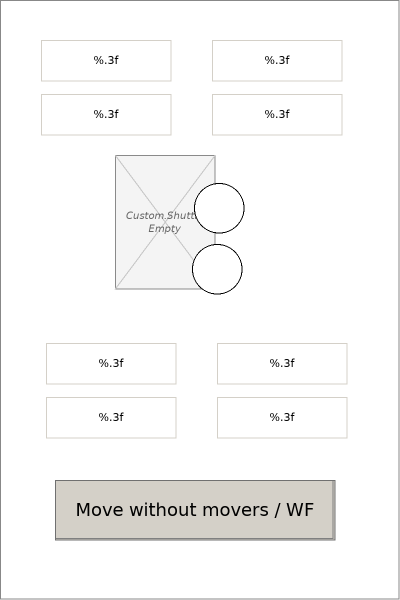
VISUALIZATION VISU_ST140  // 400x600
    Image (115,155 100x134), angle 90, invisible if: NOT __ISVALIDREF(GVL.st140_aut._Mover), image: Custom.Shuttle Empty
    Button (55,480 280x60), "Move without movers / WF", colour toggle: HMI.bArForceCyclusState[StationList_e.ST140]
        tap HMI.btArForceCyclus[StationList_e.ST140].button
    Ellipse (194,183 50x50)
    Ellipse (192,244 50x50)
    Textfield (41,40 130x41), "%.3f"
    Textfield (212,40 130x41), "%.3f"
    Textfield (212,94 130x41), "%.3f"
    Textfield (46,343 130x41), "%.3f"
    Textfield (217,343 130x41), "%.3f"
    Textfield (217,397 130x41), "%.3f"
    Textfield (41,94 130x41), "%.3f"
    Textfield (46,397 130x41), "%.3f"
END_VISUALIZATION

(* stored: Version 1.1.0.1, ProductVersion 3.1.4024.6
   Visu VISU_ST140: Id {f5c031a1-1441-4981-97ea-5c2861b68021} *)
